TYPE T_Ctrl_SIf_MOD :
STRUCT
	///configuration
	Cfg: T_Ctrl_SIf_MOD_Cfg;
	///parameter
	Par: T_Ctrl_SIf_MOD_Par;
	///current values
	Cur: T_Ctrl_SIf_MOD_Cur;
	///In: T_Ctrl_SIf_MOD_In;
	///Out: T_Ctrl_SIf_MOD_Out;
	Alm: ARRAY[1..7] OF T_Ctrl_Alm;
	
	///Data Channel from LineControl to PLC
	DtChnToPLC: T_Ctrl_SIf_MOD_DtChnToPLC;
	
	///Data Channel from PLC to LineControl
	DtChnToLine: T_Ctrl_SIf_MOD_DtChnToLine;
	
END_STRUCT
END_TYPE

(* stored: Version 1.1.0.1, ProductVersion 3.1.0.19
   DUT T_Ctrl_SIf_MOD: Id {25c02d6f-6c80-4fb0-a5bd-dc4ba1e2fdd8} *)
